% RSLogix 500 project PLC.RSS, saved by version 9.00.00.04 %
PROJECT "UNTITLED"    % processor: MicroLogix 1000 %

PROGRAM FILES
  LAD 2 "MAIN_PROG"  34 rungs
  LAD 3 "USER_FAULT"  1 rungs
  LAD 4 "HSC_INT"  1 rungs
  LAD 5 "STI_INT"  1 rungs
  LAD 6, 7, 8, 9, 10, 11, 12, 13, 14, 15, 16: only END

DATA FILES
  O0 OUTPUT  1 elements
  I1 INPUT  2 elements
  S2 STATUS  33 elements
  B3 BINARY  32 elements
  T4 TIMER  40 elements
  C5 COUNTER  32 elements
  R6 CONTROL  16 elements
  N7 INTEGER  105 elements

LADDER 2 "MAIN_PROG"
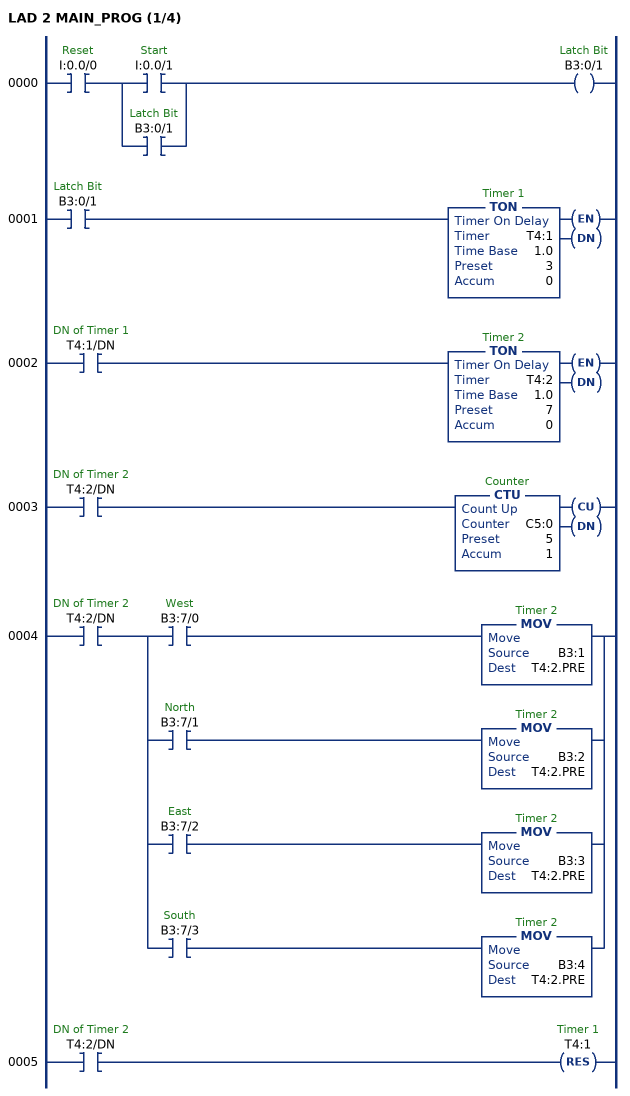
% Rung: 0 %
SOR XIC I:0.0/0 BST XIC I:0.0/1 NXB XIC B3:0/1 BND OTE B3:0/1 EOR
%   I:0.0/0  "Reset" %
%   I:0.0/1  "Start" %
%   B3:0/1  "Latch Bit" %
% Rung: 1 %
SOR XIC B3:0/1 TON T4:1 1.0 3 0 EOR
%   B3:0/1  "Latch Bit" %
%   T4:1  "Timer 1" %
% Rung: 2 %
SOR XIC T4:1/DN TON T4:2 1.0 7 0 EOR
%   T4:1/DN  "DN of Timer 1" %
%   T4:2  "Timer 2" %
% Rung: 3 %
SOR XIC T4:2/DN CTU C5:0 5 1 EOR
%   T4:2/DN  "DN of Timer 2" %
%   C5:0  "Counter" %
% Rung: 4 %
SOR XIC T4:2/DN BST XIC B3:7/0 MOV B3:1 T4:2.PRE NXB BST XIC B3:7/1 MOV B3:2 T4:2.PRE NXB BST XIC B3:7/2 MOV B3:3 T4:2.PRE NXB XIC B3:7/3 MOV B3:4 T4:2.PRE BND BND BND EOR
%   T4:2/DN  "DN of Timer 2" %
%   B3:7/0  "West" %
%   T4:2  "Timer 2" %
%   B3:7/1  "North" %
%   B3:7/2  "East" %
%   B3:7/3  "South" %
% Rung: 5 %
SOR XIC T4:2/DN RES T4:1 EOR
%   T4:2/DN  "DN of Timer 2" %
%   T4:1  "Timer 1" %

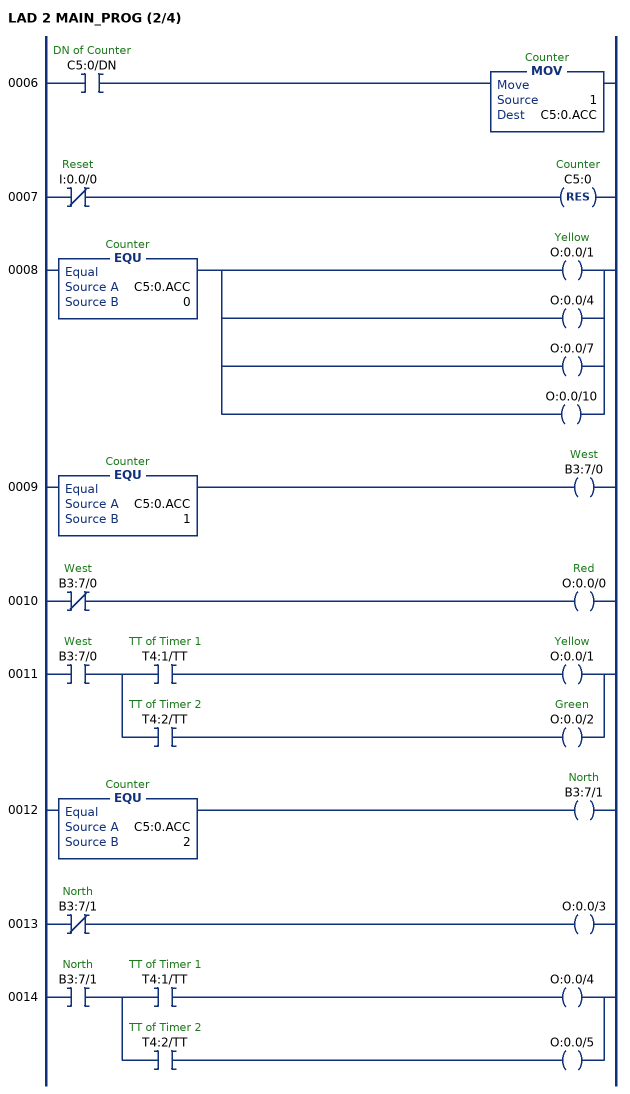
% Rung: 6 %
SOR XIC C5:0/DN MOV 1 C5:0.ACC EOR
%   C5:0/DN  "DN of Counter" %
%   C5:0  "Counter" %
% Rung: 7 %
SOR XIO I:0.0/0 RES C5:0 EOR
%   I:0.0/0  "Reset" %
%   C5:0  "Counter" %
% Rung: 8 %
SOR EQU C5:0.ACC 0 BST OTE O:0.0/1 NXB BST OTE O:0.0/4 NXB BST OTE O:0.0/7 NXB OTE O:0.0/10 BND BND BND EOR
%   C5:0  "Counter" %
%   O:0.0/1  "Yellow" %
% Rung: 9 %
SOR EQU C5:0.ACC 1 OTE B3:7/0 EOR
%   C5:0  "Counter" %
%   B3:7/0  "West" %
% Rung: 10 %
SOR XIO B3:7/0 OTE O:0.0/0 EOR
%   B3:7/0  "West" %
%   O:0.0/0  "Red" %
% Rung: 11 %
SOR XIC B3:7/0 BST XIC T4:1/TT OTE O:0.0/1 NXB XIC T4:2/TT OTE O:0.0/2 BND EOR
%   B3:7/0  "West" %
%   T4:1/TT  "TT of Timer 1" %
%   O:0.0/1  "Yellow" %
%   T4:2/TT  "TT of Timer 2" %
%   O:0.0/2  "Green" %
% Rung: 12 %
SOR EQU C5:0.ACC 2 OTE B3:7/1 EOR
%   C5:0  "Counter" %
%   B3:7/1  "North" %
% Rung: 13 %
SOR XIO B3:7/1 OTE O:0.0/3 EOR
%   B3:7/1  "North" %
% Rung: 14 %
SOR XIC B3:7/1 BST XIC T4:1/TT OTE O:0.0/4 NXB XIC T4:2/TT OTE O:0.0/5 BND EOR
%   B3:7/1  "North" %
%   T4:1/TT  "TT of Timer 1" %
%   T4:2/TT  "TT of Timer 2" %

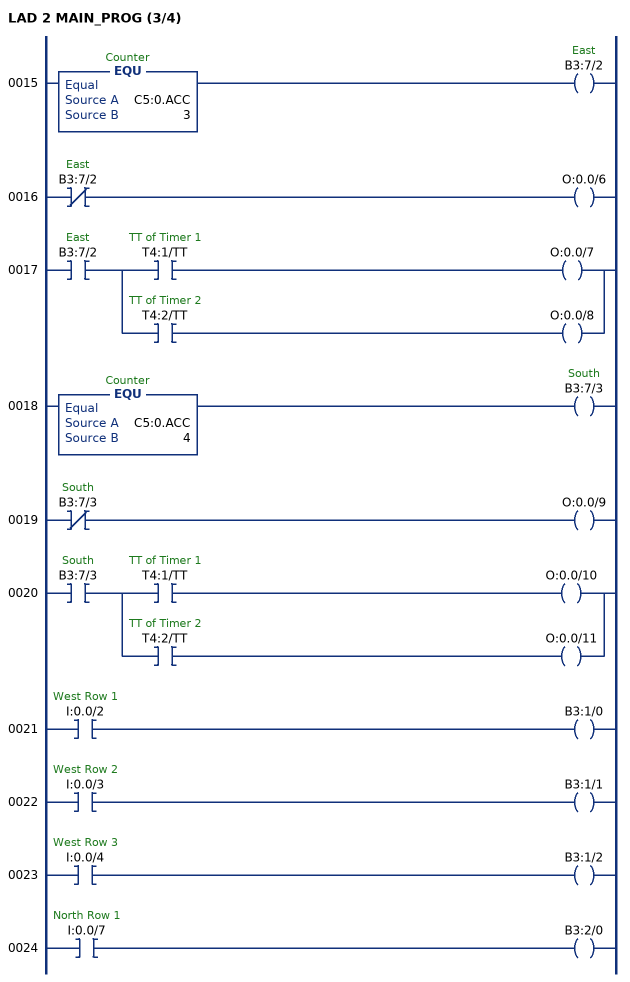
% Rung: 15 %
SOR EQU C5:0.ACC 3 OTE B3:7/2 EOR
%   C5:0  "Counter" %
%   B3:7/2  "East" %
% Rung: 16 %
SOR XIO B3:7/2 OTE O:0.0/6 EOR
%   B3:7/2  "East" %
% Rung: 17 %
SOR XIC B3:7/2 BST XIC T4:1/TT OTE O:0.0/7 NXB XIC T4:2/TT OTE O:0.0/8 BND EOR
%   B3:7/2  "East" %
%   T4:1/TT  "TT of Timer 1" %
%   T4:2/TT  "TT of Timer 2" %
% Rung: 18 %
SOR EQU C5:0.ACC 4 OTE B3:7/3 EOR
%   C5:0  "Counter" %
%   B3:7/3  "South" %
% Rung: 19 %
SOR XIO B3:7/3 OTE O:0.0/9 EOR
%   B3:7/3  "South" %
% Rung: 20 %
SOR XIC B3:7/3 BST XIC T4:1/TT OTE O:0.0/10 NXB XIC T4:2/TT OTE O:0.0/11 BND EOR
%   B3:7/3  "South" %
%   T4:1/TT  "TT of Timer 1" %
%   T4:2/TT  "TT of Timer 2" %
% Rung: 21 %
SOR XIC I:0.0/2 OTE B3:1/0 EOR
%   I:0.0/2  "West Row 1" %
% Rung: 22 %
SOR XIC I:0.0/3 OTE B3:1/1 EOR
%   I:0.0/3  "West Row 2" %
% Rung: 23 %
SOR XIC I:0.0/4 OTE B3:1/2 EOR
%   I:0.0/4  "West Row 3" %
% Rung: 24 %
SOR XIC I:0.0/7 OTE B3:2/0 EOR
%   I:0.0/7  "North Row 1" %

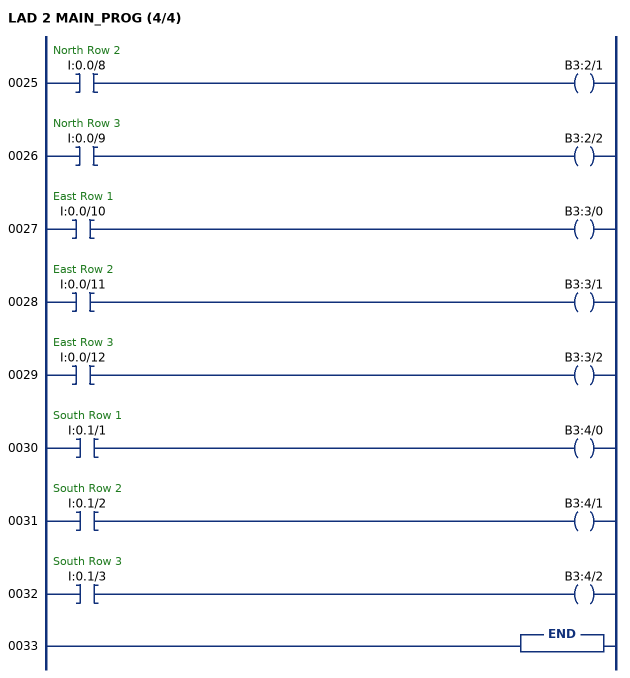
% Rung: 25 %
SOR XIC I:0.0/8 OTE B3:2/1 EOR
%   I:0.0/8  "North Row 2" %
% Rung: 26 %
SOR XIC I:0.0/9 OTE B3:2/2 EOR
%   I:0.0/9  "North Row 3" %
% Rung: 27 %
SOR XIC I:0.0/10 OTE B3:3/0 EOR
%   I:0.0/10  "East Row 1" %
% Rung: 28 %
SOR XIC I:0.0/11 OTE B3:3/1 EOR
%   I:0.0/11  "East Row 2" %
% Rung: 29 %
SOR XIC I:0.0/12 OTE B3:3/2 EOR
%   I:0.0/12  "East Row 3" %
% Rung: 30 %
SOR XIC I:0.1/1 OTE B3:4/0 EOR
%   I:0.1/1  "South Row 1" %
% Rung: 31 %
SOR XIC I:0.1/2 OTE B3:4/1 EOR
%   I:0.1/2  "South Row 2" %
% Rung: 32 %
SOR XIC I:0.1/3 OTE B3:4/2 EOR
%   I:0.1/3  "South Row 3" %
% Rung: 33 %
SOR END EOR

DATA TABLE (non-zero values as saved)
DATA T4
% .PRE .ACC %
% T4:1 % 3 0
% T4:2 % 7 0
DATA C5
% .PRE .ACC %
% C5:0 % 5 1
